PROGRAM PRG_GetItemAIManual
VAR
	sFullCode		: T_MaxString;
	eCodeType		: CODE.E_CodeAI;
	stCodeInfo		: CODE.ST_CodeInfo;
	
	sF_GetItemAI	: T_MaxString;

END_VAR

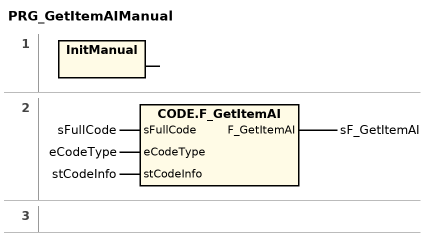
// NETWORK 1
InitManual();

// NETWORK 2
sF_GetItemAI := CODE.F_GetItemAI(sFullCode := sFullCode, eCodeType := eCodeType, stCodeInfo := stCodeInfo);

// NETWORK 3

ACTION InitManual:

sFullCode	:= '(01)17501031711052(21)86174He081137058500(240)10108245(10)86352024(91)5304012';
stCodeInfo.eCodeType	:= CODE.E_CodeType.E_CASE;

	
//eCodeType	:= CODE.E_CodeAI.GTIN;
eCodeType	:= CODE.E_CodeAI.SERIAL;
//eCodeType	:= CODE.E_CodeAI.RSKU;
//eCodeType	:= CODE.E_CodeAI.BATCH;
//eCodeType	:= CODE.E_CodeAI.PO;


// GTIN 
	stCodeInfo.stGTIN.sStartAI := '(01)';
	stCodeInfo.stGTIN.sEndAI := '(';
	stCodeInfo.stGTIN.nCodeLength := 14;
	stCodeInfo.stGTIN.nCodeStartPos := 0;	
	
// SERIAL	
	stCodeInfo.stSerialCode.sStartAI := '(21)';
	stCodeInfo.stSerialCode.sEndAI := '(';
	stCodeInfo.stSerialCode.nCodeLength := 19;
	stCodeInfo.stSerialCode.nCodeStartPos := 0;	
	
// RSKU
	stCodeInfo.stRSKU.sStartAI := '(240)';
	stCodeInfo.stRSKU.sEndAI := '(';
	stCodeInfo.stRSKU.nCodeLength := 8;
	stCodeInfo.stRSKU.nCodeStartPos := 0;	
	
// BATCH
	stCodeInfo.stBatchID.sStartAI := '(10)';
	stCodeInfo.stBatchID.sEndAI := '(';
	stCodeInfo.stBatchID.nCodeLength := 8;
	stCodeInfo.stBatchID.nCodeStartPos := 0;	
	
// PRODUCTION ORDER
	stCodeInfo.stProductionOrder.sStartAI := '(91)';
	stCodeInfo.stProductionOrder.sEndAI := '(';
	stCodeInfo.stProductionOrder.nCodeLength := 7;
	stCodeInfo.stProductionOrder.nCodeStartPos := 0;	



stCodeInfo.nMinLength 		:= 10;
stCodeInfo.nEntireLength	:= 77;
stCodeInfo.nNumberOfAIs		:= 5;
END_ACTION

END_PROGRAM

(* stored: Version 1.1.0.1
   POU PRG_GetItemAIManual: Id {dff04167-7d63-4e54-ae52-95120ff519c5}, SpecialFunc None
   Action InitManual: Id {82e374ac-3a1c-4ce3-97a1-fb1ecbadc4a3} *)
